// Gets the lower bound index of the array of specified type.
FUNCTION F_GetXWordArrayLowerBound : T_Position // The lower bound index of the specified array.
VAR_IN_OUT
	arArray : ARRAY[*] OF __XWORD; // The array to query.
END_VAR

F_GetXWordArrayLowerBound := LOWER_BOUND(arArray, 1);

END_FUNCTION

(* stored: Version 1.1.0.1
   POU F_GetXWordArrayLowerBound: Id {13c6a45b-a1da-08df-30b8-d0e7d181024f}, SpecialFunc None *)
